// Mitsubishi GX Works2 project: contador   PLC: Q03UDV

PROGRAM MAIN
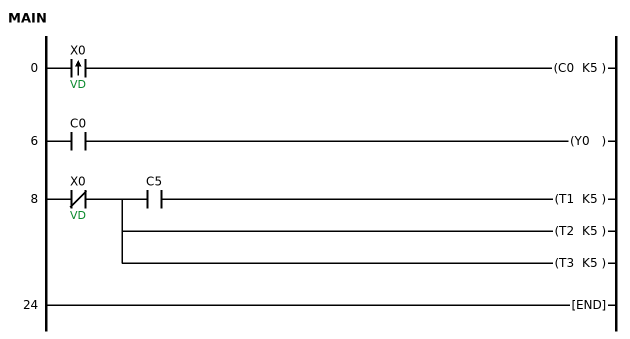
0     LDP     X0  ; VD
      OUT     C0 K5
6     LD      C0
      OUT     Y0
8     LDI     X0  ; VD
      MPS
      AND     C5
      OUT     T1 K5
      MPP
      OUT     T2 K5
      OUT     T3 K5
24    END
END_PROGRAM
